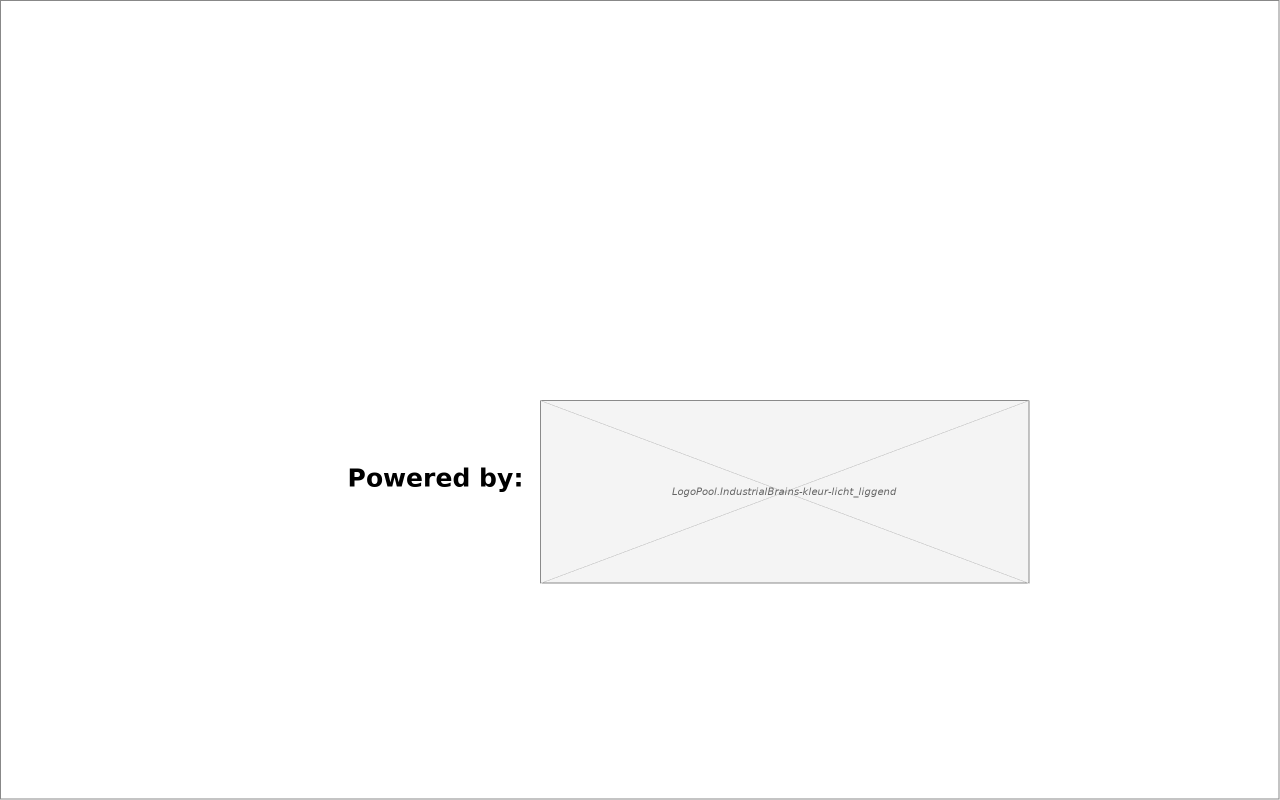
VISUALIZATION Idle  // 1280x800
    Image (540,400 489x183), image: LogoPool.IndustrialBrains-kleur-licht_liggend
    Label (340,400 200x155), "Powered by:"
END_VISUALIZATION

(* stored: Version 1.1.0.1, ProductVersion 3.1.4024.11
   Visu Idle: Id {9c0dfbb2-ead7-41c1-9ffd-e66a861a7940} *)
